PROGRAM motor_vfd_control
VAR PERSISTENT
	//Example motor starter block.  
	u_3112 : motor_vfd;
END_VAR

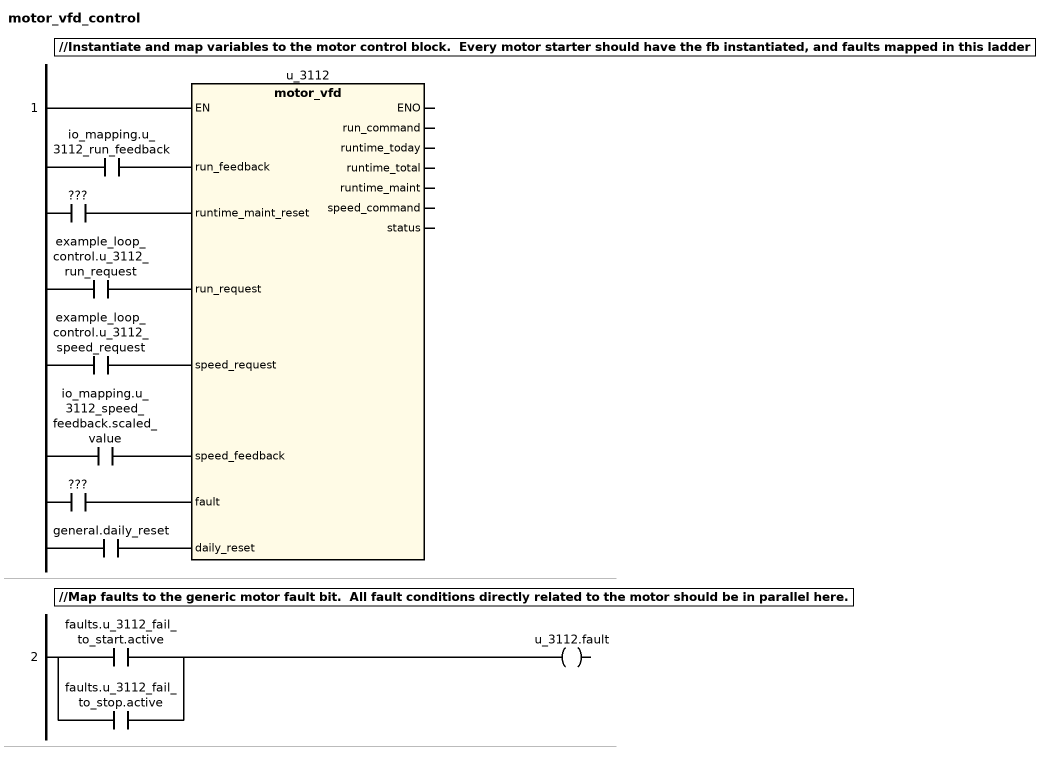
// NETWORK 1
// label: //Instantiate and map variables to the motor control block.  Every motor starter should have the fb instantiated, and faults mapped in this ladder
u_3112(
    run_feedback := io_mapping.u_3112_run_feedback,
    run_request := example_loop_control.u_3112_run_request,
    speed_request := example_loop_control.u_3112_speed_request,
    speed_feedback := io_mapping.u_3112_speed_feedback.scaled_value,
    daily_reset := general.daily_reset); // motor_vfd

// NETWORK 2
// label: //Map faults to the generic motor fault bit.  All fault conditions directly related to the motor should be in parallel here.
u_3112.fault := faults.u_3112_fail_to_start.active OR faults.u_3112_fail_to_stop.active;

END_PROGRAM

(* stored: Version 1.1.0.1, ProductVersion 3.1.4024.12
   POU motor_vfd_control: Id {eb3dd974-08a1-4d0e-8037-d05478653eb3}, SpecialFunc None *)
